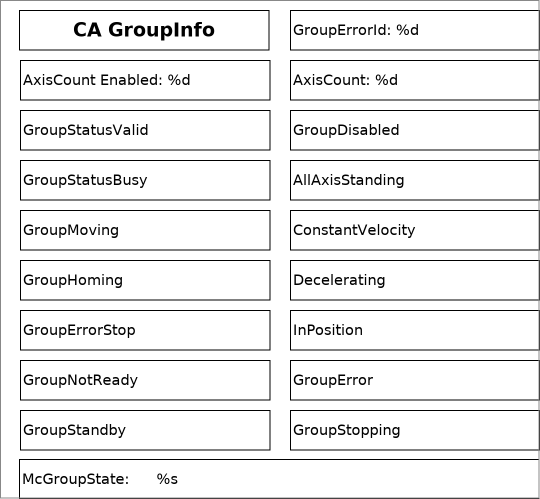
VISUALIZATION GROUP_VISU  // 540x499
VAR_IN_OUT
	stGroupInfo   : ST_GROUP_INFO;
  sGroupState   : string(60);
END_VAR
    Rectangle (20,110 250x40), "GroupStatusValid", colour toggle: stGroupInfo.GroupStatusValid
    Rectangle (20,160 250x40), "GroupStatusBusy", colour toggle: stGroupInfo.GroupStatusBusy
    Rectangle (20,210 250x40), "GroupMoving", colour toggle: stGroupInfo.GroupMoving
    Rectangle (20,260 250x40), "GroupHoming", colour toggle: stGroupInfo.GroupHoming
    Rectangle (20,310 250x40), "GroupErrorStop", colour toggle: stGroupInfo.GroupErrorStop
    Rectangle (20,360 250x40), "GroupNotReady", colour toggle: stGroupInfo.GroupNotReady
    Rectangle (20,410 250x40), "GroupStandby", colour toggle: stGroupInfo.GroupStandby
    Rectangle (290,410 250x40), "GroupStopping", colour toggle: stGroupInfo.GroupStopping
    Rectangle (290,110 250x40), "GroupDisabled", colour toggle: stGroupInfo.GroupDisabled
    Rectangle (290,160 250x40), "AllAxisStanding", colour toggle: stGroupInfo.AllAxesStanding
    Rectangle (290,210 250x40), "ConstantVelocity", colour toggle: stGroupInfo.ConstantVelocity
    Rectangle (290,260 250x40), "Decelerating", colour toggle: stGroupInfo.Decelerating
    Rectangle (290,310 250x40), "InPosition", colour toggle: stGroupInfo.InPosition
    Rectangle (290,360 250x40), "GroupError", colour toggle: stGroupInfo.GroupError
    Rectangle (290,10 250x40), "GroupErrorId: %d", text variable: stGroupInfo.GroupErrorId
    Rectangle (290,60 250x40), "AxisCount: %d", text variable: stGroupInfo.AxisCount
    Rectangle (19,459 520x40), "McGroupState: %s", text variable: sGroupState
    Rectangle (19,10 250x40), "CA GroupInfo"
    Rectangle (20,60 250x40), "AxisCount Enabled: %d", text variable: stGroupInfo.AxisCountEnabled
END_VISUALIZATION

(* stored: Version 1.1.0.1
   Visu GROUP_VISU: Id {80965c1a-a8d0-4832-8bac-c39709da9df2} *)
